FUNCTION_BLOCK PUBLIC PAEContactor EXTENDS PAESensorDigital
VAR_INPUT
END_VAR
VAR_OUTPUT
END_VAR
VAR
END_VAR

END_FUNCTION_BLOCK

(* stored: Version 1.1.0.1, ProductVersion 3.1.4020.6
   POU PAEContactor: Id {c9cf3ca8-787e-49d4-999d-388e14eeda78}, SpecialFunc None *)
